{attribute 'qualified_only'}
VAR_GLOBAL
	levitation_active:		BOOL;
	levitation_fault: 		BOOL;
	//DC link voltages
	drive_voltages: INT;
END_VAR

(* stored: Version 1.1.0.1
   GVL GVL_Levi: Id {d4dca03b-650a-425c-b19f-85a72034f677} *)
